// TIA Portal project "MonitoringPLCs" (V12)

(* hardware
DEVICE "S7-1200 station_1"  SIMATIC 1200-Station
   slot 0: "S7-1200 rack"  Rack  V1.0
   slot 1: "PLC_1"  CPU 1212C DC/DC/Rly  6ES7 212-1HD30-0XB0  V2.2
*)

// ===== PLC "PLC_1"  CPU 1212C DC/DC/Rly =====

VAR_GLOBAL   // PLC tag table "AcceleratedChamberIOs"
   "TemperatureAlarm" AT %I0.0 : Bool;
   "HumidityAlarm" AT %I0.1 : Bool;
END_VAR

VAR_GLOBAL   // PLC tag table "LongtermChamberIOs"
   "TemperatureAlarm(1)" AT %I0.2 : Bool;
   "HumidityAlarm(1)" AT %I0.3 : Bool;
END_VAR

VAR_GLOBAL   // PLC tag table "Alarms"
   "AlarmChambers" AT %Q0.0 : Bool;
   "SilentAlarm" AT %Q0.1 : Bool;
END_VAR

ORGANIZATION_BLOCK "Main"   // OB1, FBD, ProgramCycle
TITLE = "Main Program Sweep (Cycle)"
{ S7_Optimized_Access := 'FALSE' }
VERSION : 0.1
BEGIN

REGION Network 1
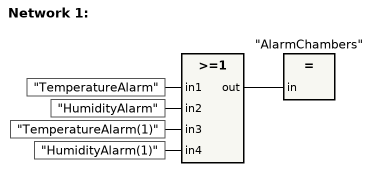
   "AlarmChambers" := "TemperatureAlarm" OR "HumidityAlarm" OR "TemperatureAlarm(1)" OR "HumidityAlarm(1)";
END_REGION
END_ORGANIZATION_BLOCK